FUNCTION_BLOCK Random
VAR_INPUT
	iMinVal	: INT;
	iMaxVal	: INT;
END_VAR
VAR_OUTPUT
	o_iResult : INT;
END_VAR
VAR
	lrMidValue : LREAL;
	iMidValue : INT;
	drand		: drand;
END_VAR

drand(Seed := 0,Num => lrMidValue);

lrMidValue := lrMidValue * 10;
iMidValue := LREAL_TO_INT(lrMidValue);

IF iMidValue > iMinVal AND iMidValue < iMaxVal THEN
	o_iResult := iMidValue;
END_IF

END_FUNCTION_BLOCK

(* stored: Version 1.1.0.1, ProductVersion 3.1.4024.13
   POU Random: Id {7d49a695-f630-4a60-accd-411f2f197065}, SpecialFunc None *)
